Universal Robots PolyScope program: z_force.urp

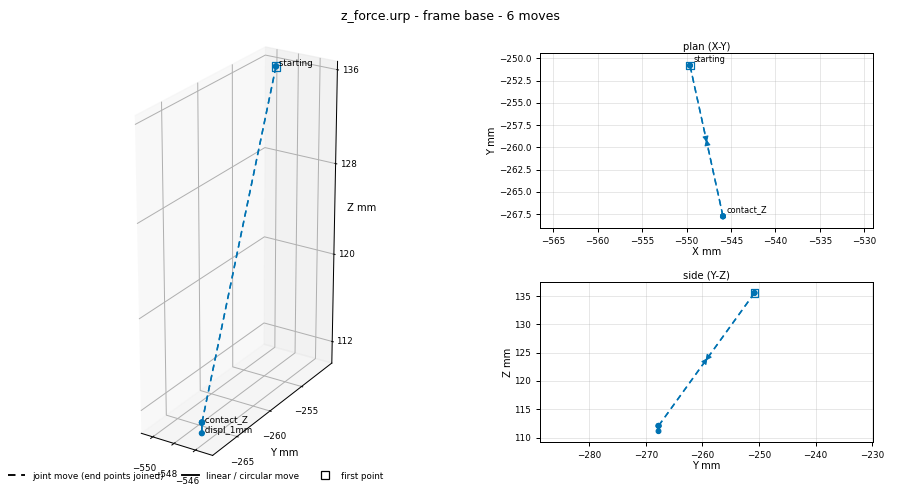
[picture p0: tool path of z_force.urp in frame base, 6 of 6 moves have a stored position in this frame; points joined in program order, loops and branches not executed]
Program z_force_mh (installation=weiss_default directory=/programs/usbdisk_0/Max_MA/new folder createdIn=5.12.4 lastSavedIn=5.14.3 robotSerialNumber=20235500024)
Calibrated DH parameters: a=[0.000122, -0.425124, -0.373197, -0.000038, 0.000163, 0]; d=[0.162581, -17.281615, 1.061906, 16.353116, 0.099729, 0.099553]; alpha=[1.570231, 0.000934, 0.007511, 1.569966, -1.569202, 0]; deltaTheta=[0, -0.037947, -0.277584, 0.315538, 0.000001, -0.000001]
InitVariablesNode
BeforeStart
  Script: socket_close("DataSocket")
  Script: connected = socket_open("192.168.100.0",30000,"DataSocket")
  force_measure := False
  If connected ≟  False (checkContinuously=true)
    Halt
Robot Program (runOnlyOnce=true)
  MoveJ speed 60 deg/s, acceleration 80 deg/s^2 (useActiveTCP=true) feature=Base
    Waypoint starting: TCP in base x=-549.607 y=-250.796 z=135.55 mm, rx=-3.1224 ry=-0.3459 rz=-0.0014 rad; joints [11.857, -67.298, 101.17, -123.73, -89.599, 89.327] deg; TCP offset x=0 y=0 z=100 mm, rx=0 ry=0 rz=0 rad
    SuppressedNode
      Set DigitalOutput pin=digital_out[0]; digitalValue=1
    Timer (action=Start) variable(name=timer_1)
    Timer (action=Start) variable(name=timer_3)
    Waypoint contact_Z: TCP in base x=-545.899 y=-267.745 z=112.074 mm, rx=-3.1223 ry=-0.3459 rz=-0.0006 rad; joints [13.535, -64.985, 101.826, -126.73, -89.611, 91.029] deg
    force_measure := True
    Loop Counting (count=10) loopVariable(name=Loop_3)
      MoveL speed 1 mm/s, acceleration 600 mm/s^2 (useActiveTCP=true) feature=Base
        Waypoint displ_1mm: TCP in base x=-545.911 y=-267.752 z=111.127 mm, rx=-3.1224 ry=-0.3458 rz=-0.0005 rad; joints [13.534, -64.906, 101.877, -126.863, -89.607, 91.033] deg
        Waypoint contact_Z: TCP in base x=-545.899 y=-267.745 z=112.074 mm, rx=-3.1223 ry=-0.3459 rz=-0.0006 rad; joints [13.535, -64.985, 101.826, -126.73, -89.611, 91.029] deg
    force_measure := False
    Waypoint contact_Z: TCP in base x=-545.899 y=-267.745 z=112.074 mm, rx=-3.1223 ry=-0.3459 rz=-0.0006 rad; joints [13.535, -64.985, 101.826, -126.73, -89.611, 91.029] deg
    Wait Sleep waitTime=2
    Timer (action=Stop) variable=timer_3
    Timer (action=Reset) variable=timer_3
    SuppressedNode
      Wait Sleep waitTime=5
    Timer (action=Stop) variable=timer_1
    Waypoint starting: TCP in base x=-549.607 y=-250.796 z=135.55 mm, rx=-3.1224 ry=-0.3459 rz=-0.0014 rad; joints [11.857, -67.298, 101.17, -123.73, -89.599, 89.327] deg
Thread Thread_1 (runOnlyOnce=false)
  If force_measure ≟ True
    counter := 1
    SuppressedNode
      Wait Sleep waitTime=1
    Timer (action=Reset) variable(name=timer_2)
    Timer (action=Start) variable=timer_2
    Loop While (checkContinuously=true) expression=force_measure ≟  True
      force_value := get_tcp_force()
      pos_value := get_actual_tcp_pose()
      SuppressedNode
        msg_out := [timer_2,force_value[0],force_value[1],force_value[2],force_value[3],force_value[4],force_value[5]]
      msg_out := [timer_2,force_value[0],force_value[1],force_value[2],force_value[3],force_value[4],force_value[5],pos_value[0],pos_value[1],pos_value[2],pos_value[3],pos_value[4],pos_value[5]]
      Script: socket_send_string(msg_out,"DataSocket")
      SuppressedNode
        Script: data = socket_read_ascii_float(1,"DataSocket")
      SuppressedNode
        screw_force_lim := data[1]
      counter := counter + 1
      Wait Sleep waitTime=0.02
    Script: socket_send_string("end","DataSocket")
    Wait Sleep waitTime=0.01
    Script: socket_close("DataSocket")
    Timer (action=Stop) variable=timer_2
SuppressedNode
  Thread Thread_2 (runOnlyOnce=false)
    URCap Gripper Activate (Robotiq_Grippers, Robotiq Inc.) dataModel(ResetAndActivateKey=true)
    URCap GRIPKIT Reference (GRIPKIT by Weiss Robotics, Weiss Robotics GmbH & Co. KG) dataModel(reference1=true)
